// TIA Portal V21 export
VAR_GLOBAL   // PLC tag table "K_TipoComunicazione"
END_VAR
VAR_GLOBAL CONSTANT   // user constants
   K_TipoComunicazione_Digitale : Int := 0;
   K_TipoComunicazione_GetPut : Int := 1;
   K_TipoComunicazione_OpcUa : Int := 2;
END_VAR
